// TIA Portal V19 export
TYPE "Positioning_DOL_Machine_DataOut"
// stored: Access Published
   STRUCT
      Fan_M_Contactor : Bool;
   END_STRUCT;
END_TYPE
